{attribute 'linkalways'} 
{attribute 'no_explicit_call' := 'This FB is a CLASS and must be accessed using methods or properties'}
{attribute 'enable_dynamic_creation'}
FUNCTION_BLOCK FINAL Node_DELETE EXTENDS Node
VAR
	str : _STRING('');
    len : _INT(0);
	pos : _INT(0);
	out : _STRING('');
END_VAR

METHOD PUBLIC  Clone : I_Node
VAR
	pNode : POINTER TO Node_DELETE;
END_VAR
pNode := __NEW(Node_DELETE);
Clone := pNode^;
END_METHOD

METHOD FB_init : BOOL
VAR_INPUT
	bInitRetains : BOOL; // if TRUE, the retain variables are initialized (warm start / cold start)
	bInCopyCode : BOOL;  // if TRUE, the instance afterwards gets moved into the copy code (online change)
END_VAR
AddParameter('str', str);
AddParameter('len', len);
AddParameter('pos', pos);
AddOutput('out', out);
END_METHOD

METHOD PROTECTED OnExecute
VAR
END_VAR
out.Value := DELETE(str.Value, len.Value, pos.Value);
END_METHOD

END_FUNCTION_BLOCK

(* stored: Version 1.1.0.1, ProductVersion 3.1.4026.18
   POU Node_DELETE: Id {e853047d-7824-06d6-1447-2d242dc7cc87}, SpecialFunc None
   Folder Constructor: Id {a2e83de6-b1e1-0abb-11a3-1f1c382311e8}
   Method Clone: Id {124137c3-be1c-09a0-15e4-1a5530d7187f}
   Method FB_init: Id {5c46fec6-8c9d-0f8c-29df-c4ec4c9f5b37}
   Method OnExecute: Id {d0055374-9099-0987-003a-3a251728d149} *)
